TYPE ST_InputsInOutFeed :
STRUCT	
	HW		: ST_HW_InputsInOutFeed;
	Ctrl	: ST_CtrlInInOutFeed;
END_STRUCT
END_TYPE

(* stored: Version 1.1.0.1, ProductVersion 3.1.4024.9
   DUT ST_InputsInOutFeed: Id {b36b2c4f-5582-408b-b2f4-0a40c1e28b3e} *)
